// TIA Portal V15.1 export
// export: Created 2024-05-17T05:38:25.0394774Z, ExportSetting WithDefaults, DisplayName Totally Integrated Automation Portal, DisplayVersion V15.1 Update 5, DisplayName TIA Portal Openness, DisplayVersion V15.1 Update 5, DisplayName SINAMICS Startdrive Advanced, DisplayVersion V15.1, DisplayName G130, G150, S120, S150, SINAMICS MV, S210, DisplayVersion V15.1, DisplayName G110M, G120, G120C, G120D, G120P, DisplayVersion V15.1, DisplayName STEP 7 Professional, DisplayVersion V15.1 Update 5, DisplayName STEP 7 Safety, DisplayVersion V15.1, DisplayName WinCC Professional, DisplayVersion V15.1 Update 5, DisplayName SIMATIC Visualization Architect, DisplayVersion V15.1
FUNCTION_BLOCK "LGenHooterFlash"   // FB1007, FBD
TITLE = LGenHootFlash
{ S7_Optimized_Access := 'FALSE' }
AUTHOR : VCG
FAMILY : VCGGen
VERSION : 1.0
// ==============================================================================
// FB 
// ==============================================================================
// stored: AutoNumber false, IsIECCheckEnabled false, SetENOAutomatically False, UDAEnableTagReadback false
   VAR_INPUT
      I_Lamptest { ExternalAccessible := 'False'; ExternalVisible := 'False'; ExternalWritable := 'False'} : Bool;   // Summation of lamptest buttons
      I_GenResetAlarm { ExternalAccessible := 'False'; ExternalVisible := 'False'; ExternalWritable := 'False'} : Bool;   // General reset alarm
      I_GenAlarmA { ExternalAccessible := 'False'; ExternalVisible := 'False'; ExternalWritable := 'False'} : Bool;   // General Alarm A active
      I_GenAlarmB { ExternalAccessible := 'False'; ExternalVisible := 'False'; ExternalWritable := 'False'} : Bool;   // General Alarm B active
      I_GenAlarmC { ExternalAccessible := 'False'; ExternalVisible := 'False'; ExternalWritable := 'False'} : Bool;   // General Alarm C active
      I_HardwareAlarm { ExternalAccessible := 'False'; ExternalVisible := 'False'; ExternalWritable := 'False'} : Bool;   // Safety circuit hardware Alarm active
      I_GenWarningStart { ExternalAccessible := 'False'; ExternalVisible := 'False'; ExternalWritable := 'False'} : Bool;   // Warning start from station
   END_VAR
   VAR_OUTPUT
      O_HooterAK { ExternalAccessible := 'False'; ExternalVisible := 'False'; ExternalWritable := 'False'} : Bool;   // Steering for hooter AK
      O_HooterAS1 { ExternalAccessible := 'False'; ExternalVisible := 'False'; ExternalWritable := 'False'} : Bool;   // Steering for hooter AS1
      O_HooterAS2 { ExternalAccessible := 'False'; ExternalVisible := 'False'; ExternalWritable := 'False'} : Bool;   // Steering for hooter AS2
      O_FlashAK { ExternalAccessible := 'False'; ExternalVisible := 'False'; ExternalWritable := 'False'} : Bool;   // Steering for flashlight AK
      O_FlashAS1 { ExternalAccessible := 'False'; ExternalVisible := 'False'; ExternalWritable := 'False'} : Bool;   // Steering for flashlight AS1
      O_FlashAS2 { ExternalAccessible := 'False'; ExternalVisible := 'False'; ExternalWritable := 'False'} : Bool;   // Steering for flashlight AS2
   END_VAR
   VAR DB_SPECIFIC
      HooterForAlmAB { ExternalAccessible := 'False'; ExternalVisible := 'False'; ExternalWritable := 'False'} : Bool;   // Hooter activation for fault A or B
      HooterForWarnSt { ExternalAccessible := 'False'; ExternalVisible := 'False'; ExternalWritable := 'False'} : Bool;   // Hooter activation for warningstart
      DelayTimeElapsed { ExternalAccessible := 'False'; ExternalVisible := 'False'; ExternalWritable := 'False'} : Bool;   // Timer result (on during max 1 hour)
      ResetDone { ExternalAccessible := 'False'; ExternalVisible := 'False'; ExternalWritable := 'False'} : Bool;   // Reset done
      DelayTimerValue { ExternalAccessible := 'False'; ExternalVisible := 'False'; ExternalWritable := 'False'} : DInt;   // Delay Timer elapsed
   END_VAR
   VAR
      DelayTimer { ExternalAccessible := 'False'; ExternalVisible := 'False'; ExternalWritable := 'False'; S7_SetPoint := 'True'} : "LTimer";
   END_VAR
BEGIN

REGION Network 1: *** 1 - Inputs *** Timer for maximum 1 hour operation of the hooter
   // Timer for maximum 1 hour operation of the hooter
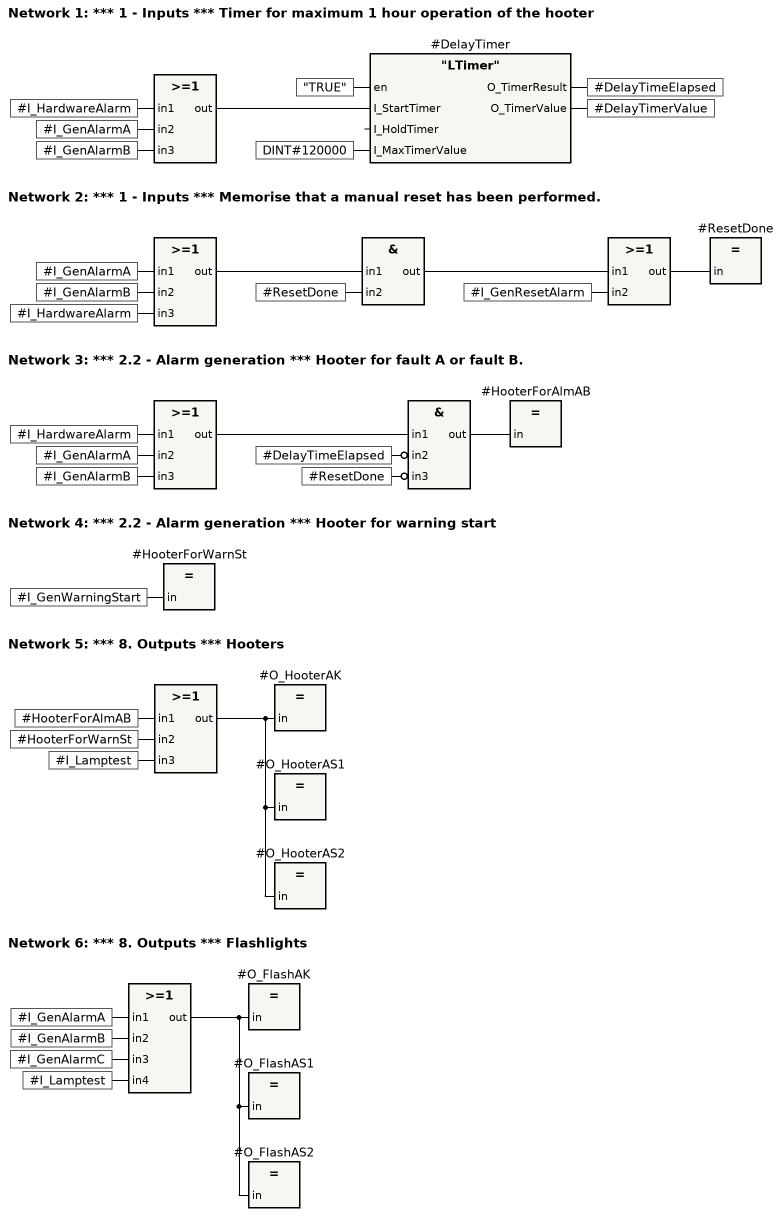
   IF "TRUE" THEN
       #DelayTimer(I_StartTimer := #I_HardwareAlarm OR #I_GenAlarmA OR #I_GenAlarmB,   // "LTimer"
                   I_MaxTimerValue := DINT#120000,
                   O_TimerResult => #DelayTimeElapsed,
                   O_TimerValue => #DelayTimerValue);
   END_IF;
END_REGION

REGION Network 2: *** 1 - Inputs *** Memorise that a manual reset has been performed.
   // Memorise that a manual reset has been performed.
   #ResetDone := ((#I_GenAlarmA OR #I_GenAlarmB OR #I_HardwareAlarm) AND #ResetDone) OR #I_GenResetAlarm;
END_REGION

REGION Network 3: *** 2.2 - Alarm generation *** Hooter for fault A or fault B.
   // Hooter for fault A or fault B.
   // Muted after x time OR when reset button was pressed.
   #HooterForAlmAB := (#I_HardwareAlarm OR #I_GenAlarmA OR #I_GenAlarmB) AND NOT #DelayTimeElapsed AND NOT #ResetDone;
END_REGION

REGION Network 4: *** 2.2 - Alarm generation *** Hooter for warning start
   // Hooter for warning start
   #HooterForWarnSt := #I_GenWarningStart;
END_REGION

REGION Network 5: *** 8. Outputs *** Hooters
   // Hooters
   #O_HooterAK := #HooterForAlmAB OR #HooterForWarnSt OR #I_Lamptest;
   #O_HooterAS1 := #O_HooterAK;
   #O_HooterAS2 := #O_HooterAK;
END_REGION

REGION Network 6: *** 8. Outputs *** Flashlights
   // Flashlights
   #O_FlashAK := #I_GenAlarmA OR #I_GenAlarmB OR #I_GenAlarmC OR #I_Lamptest;
   #O_FlashAS1 := #O_FlashAK;
   #O_FlashAS2 := #O_FlashAK;
END_REGION
END_FUNCTION_BLOCK
